# EPICS substitutions: viocs/tb_ps/tb_psApp/Db/ch.substitutions
file "db/individual.db" {
    pattern { family, pos }
        { "CH", "03" }
}
